{attribute 'linkalways'} 
{attribute 'no_explicit_call' := 'This FB is a CLASS and must be accessed using methods or properties'}
{attribute 'enable_dynamic_creation'}
FUNCTION_BLOCK FINAL MUL_UINT EXTENDS Node
VAR
	in1 : _UINT(0);
	in2 : _UINT(0);
	out : _UINT(0);
END_VAR

METHOD PUBLIC Clone : I_Node
VAR
	pNode : POINTER TO MUL_UINT;
END_VAR
pNode := __NEW(MUL_UINT);
Clone := pNode^;
END_METHOD

METHOD FB_init : BOOL
VAR_INPUT
	bInitRetains : BOOL; // if TRUE, the retain variables are initialized (warm start / cold start)
	bInCopyCode : BOOL;  // if TRUE, the instance afterwards gets moved into the copy code (online change)
END_VAR
AddInput('in1',THIS^.in1);
AddInput('in2',THIS^.in2);
AddOutput('out', THIS^.out);
END_METHOD

METHOD PROTECTED OnExecute
VAR
END_VAR
out.Value := in1.Value * in2.Value;
END_METHOD

END_FUNCTION_BLOCK

(* stored: Version 1.1.0.1, ProductVersion 3.1.4024.15
   POU MUL_UINT: Id {867a5f0c-0c7d-42fb-af18-e0e61a696d2a}, SpecialFunc None
   Folder Constructor: Id {258d6dca-fefc-4968-b899-45fb9a96e1c3}
   Method Clone: Id {01ddc496-b9b2-43d1-9a71-48f61171cb97}
   Method FB_init: Id {0fc37c67-e0cc-4d9f-8ee9-fd3f5ba7c193}
   Method OnExecute: Id {b5dcf8a6-602a-40be-97b0-c1f8724b55b3} *)
